PROGRAM PRG_2_AT1K4
VAR
	
   {attribute 'pytmc' := 'pv: AT1K4:L2SI:'}
    {attribute 'TcLinkTo' := '
        .RTD_Axis1_1.iRaw := TIIB[AT1K4-EL3202-01]^RTD Inputs Channel 1^Value;
        .RTD_Axis1_1.bError := TIIB[AT1K4-EL3202-01]^RTD Inputs Channel 1^Status^Error;
        .RTD_Axis1_1.bUnderrange := TIIB[AT1K4-EL3202-01]^RTD Inputs Channel 1^Status^Underrange;
        .RTD_Axis1_1.bOverrange := TIIB[AT1K4-EL3202-01]^RTD Inputs Channel 1^Status^Overrange;

        .RTD_Axis1_2.iRaw := TIIB[AT1K4-EL3202-01]^RTD Inputs Channel 2^Value;
        .RTD_Axis1_2.bError := TIIB[AT1K4-EL3202-01]^RTD Inputs Channel 2^Status^Error;
        .RTD_Axis1_2.bUnderrange := TIIB[AT1K4-EL3202-01]^RTD Inputs Channel 2^Status^Underrange;
        .RTD_Axis1_2.bOverrange := TIIB[AT1K4-EL3202-01]^RTD Inputs Channel 2^Status^Overrange;


        .RTD_Axis2_1.iRaw := TIIB[AT1K4-EL3202-02]^RTD Inputs Channel 1^Value;
        .RTD_Axis2_1.bError := TIIB[AT1K4-EL3202-02]^RTD Inputs Channel 1^Status^Error;
        .RTD_Axis2_1.bUnderrange := TIIB[AT1K4-EL3202-02]^RTD Inputs Channel 1^Status^Underrange;
        .RTD_Axis2_1.bOverrange := TIIB[AT1K4-EL3202-02]^RTD Inputs Channel 1^Status^Overrange;

        .RTD_Axis2_2.iRaw := TIIB[AT1K4-EL3202-02]^RTD Inputs Channel 2^Value;
        .RTD_Axis2_2.bError := TIIB[AT1K4-EL3202-02]^RTD Inputs Channel 2^Status^Error;
        .RTD_Axis2_2.bUnderrange := TIIB[AT1K4-EL3202-02]^RTD Inputs Channel 2^Status^Underrange;
        .RTD_Axis2_2.bOverrange := TIIB[AT1K4-EL3202-02]^RTD Inputs Channel 2^Status^Overrange;


        .RTD_Axis3_1.iRaw := TIIB[AT1K4-EL3202-03]^RTD Inputs Channel 1^Value;
        .RTD_Axis3_1.bError := TIIB[AT1K4-EL3202-03]^RTD Inputs Channel 1^Status^Error;
        .RTD_Axis3_1.bUnderrange := TIIB[AT1K4-EL3202-03]^RTD Inputs Channel 1^Status^Underrange;
        .RTD_Axis3_1.bOverrange := TIIB[AT1K4-EL3202-03]^RTD Inputs Channel 1^Status^Overrange;

        .RTD_Axis3_2.iRaw := TIIB[AT1K4-EL3202-03]^RTD Inputs Channel 2^Value;
        .RTD_Axis3_2.bError := TIIB[AT1K4-EL3202-03]^RTD Inputs Channel 2^Status^Error;
        .RTD_Axis3_2.bUnderrange := TIIB[AT1K4-EL3202-03]^RTD Inputs Channel 2^Status^Underrange;
        .RTD_Axis3_2.bOverrange := TIIB[AT1K4-EL3202-03]^RTD Inputs Channel 2^Status^Overrange;


        .RTD_Axis4_1.iRaw := TIIB[AT1K4-EL3202-04]^RTD Inputs Channel 1^Value;
        .RTD_Axis4_1.bError := TIIB[AT1K4-EL3202-04]^RTD Inputs Channel 1^Status^Error;
        .RTD_Axis4_1.bUnderrange := TIIB[AT1K4-EL3202-04]^RTD Inputs Channel 1^Status^Underrange;
        .RTD_Axis4_1.bOverrange := TIIB[AT1K4-EL3202-04]^RTD Inputs Channel 1^Status^Overrange;

        .RTD_Axis4_2.iRaw := TIIB[AT1K4-EL3202-04]^RTD Inputs Channel 2^Value;
        .RTD_Axis4_2.bError := TIIB[AT1K4-EL3202-04]^RTD Inputs Channel 2^Status^Error;
        .RTD_Axis4_2.bUnderrange := TIIB[AT1K4-EL3202-04]^RTD Inputs Channel 2^Status^Underrange;
        .RTD_Axis4_2.bOverrange := TIIB[AT1K4-EL3202-04]^RTD Inputs Channel 2^Status^Overrange;

    '}
    prg_2_at1k4 : FB_SATT;
	
	 bDebug : BOOL := FALSE;
    nEnableMode: ENUM_StageEnableMode;
	
END_VAR

(* Motion *)

IF bDebug THEN
    // NEVER: checkouts with the TwinCAT NC GUI.
    nEnableMode := ENUM_StageEnableMode.NEVER;
ELSE
    // ALWAYS: want active position correction at all times
    nEnableMode := ENUM_StageEnableMode.ALWAYS;
END_IF


prg_2_at1k4(stMotion1:=Main.M1,
			stMotion2:=Main.M2,
			stMotion3:=Main.M3,
			stMotion4:=Main.M4,
			nEnableMode:= nEnableMode);

END_PROGRAM

(* stored: Version 1.1.0.1, ProductVersion 3.1.4024.3
   POU PRG_2_AT1K4: Id {015e73b3-638b-4df6-82a5-39fd68ea7458}, SpecialFunc None *)
